TYPE MC_CMD :
STRUCT
	bExe:BOOL;
	lrVelocity:LREAL;
	lrAcceleration:LREAL;
	LrDeceleration:LREAL;
	lrJerk:LREAL;
	lrDistance:LREAL;
	lrPosition:LREAL;
	EnuDirection:  MC_Direction;
	EnuBufferMode: MC_BufferMode;
	EnuOptions  :  ST_MoveOptions;
END_STRUCT
END_TYPE

(* stored: Version 1.1.0.1, ProductVersion 3.1.4024.13
   DUT MC_CMD: Id {00bc414e-9a1d-4b31-b1c9-db084bb2d153} *)
